// How to initialize plant control at declaration (Recommended workflow).
// [Hint]
// > All reference-variables are implemented to ease monitoring of relevant variables.
FUNCTION_BLOCK FB_Plt_Init1 EXTENDS FB_BA_View
VAR
   	{region 'Aggregates'}
		DmprSu_Open							: REFERENCE TO BOOL							REF= DmprSu.bOpen;
		DmprSu_Val							: REFERENCE TO REAL							REF= DmprSu.fActiveVal;
		DmprSu								: FB_TimerAggregateA						:= (iParent:=THIS^,					iLabel:=MyLabels.DmprSu);
		FanSu_Val							: REFERENCE TO UDINT						REF= FanSu.nActiveVal;
		FanSu								: FB_BA_AggregateM							:= (iParent:=THIS^,					iLabel:=MyLabels.FanSu);
			 
		DmprEx_Open							: REFERENCE TO BOOL							REF= DmprEx.bOpen;
		DmprEx_Val							: REFERENCE TO REAL							REF= DmprEx.fActiveVal;
		DmprEx								: FB_TimerAggregateA						:= (iParent:=THIS^,					iLabel:=MyLabels.DmprEx);
		FanEx_Val							: REFERENCE TO UDINT						REF= FanEx.nActiveVal;
		FanEx								: FB_BA_AggregateM							:= (iParent:=THIS^,					iLabel:=MyLabels.FanEx);
			 
		PreHtr_Proc							: REFERENCE TO BOOL							REF= PreHtr.Process.bActive;
		PreHtr_Val							: REFERENCE TO BOOL							REF= PreHtr.bActiveVal;
		PreHtr								: FB_ProcAggregateB							:= (iParent:=THIS^,					iLabel:=MyLabels.PreHtr,			Process:=(iLabel:=MyLabels.ProcPreRinse));
		Erc_Val								: REFERENCE TO BOOL							REF= Erc.bActiveVal;
		Erc									: FB_BA_AggregateB							:= (iParent:=THIS^,					iLabel:=MyLabels.Erc);
		Col_Val								: REFERENCE TO BOOL							REF= Col.bActiveVal;
		Col									: FB_BA_AggregateB							:= (iParent:=THIS^,					iLabel:=MyLabels.Col);
	{endregion}
	{region 'Plant'} 
		OpMode								: E_OpMod_AC								:= E_OpMod_AC.eOff;
		PlantCtrl_OpSta						: REFERENCE TO BOOL							REF= PlantCtrl.bOpSta;
		PlantCtrl_On						: REFERENCE TO BOOL							REF= PlantCtrl.bOn;
		PlantCtrl_PrVal						: REFERENCE TO UDINT						REF= PlantCtrl.nPresentValue;
		PlantCtrl_Step						: REFERENCE TO STRING						REF= PlantCtrl.sStep;
		PlantCtrl							: FB_BA_PlantCtrl := (
												iParent									:= THIS^,
												iLabel									:= MyLabels.PltCtrl,
												stOperation := (
													aOpMode								:= [ E_OpMod_AC.eDisturb,				E_OpMod_AC.eSmokeExtract,		E_OpMod_AC.eOff,			E_OpMod_AC.eOn,				E_OpMod_AC.eNightCool ],
													aPriority							:= [ E_BA_Priority.eCritical,			E_BA_Priority.eLifeSafety,		E_BA_Priority.eProgram,		E_BA_Priority.eProgram,		E_BA_Priority.eProgram ],
													aIgnoreFlags						:= [ E_BA_AggregateIgnoreFlags.Delay,	E_BA_AggregateIgnoreFlags.All,	0,							0,							0 ],
													aAggregates := [(
														iReference						:= DmprSu,
														aAggMode						:= [ 0,									100,							0,							100,						100 ]
													), (
														iReference						:= DmprEx,
														aAggMode						:= [ 0,									100,							0,							100,						100 ]
													), (
														iReference						:= PreHtr,
														aAggMode						:= [ E_OpMod_Binary.eOff,				E_OpMod_Binary.eOn,				E_OpMod_Binary.eOff,		E_OpMod_Binary.eOn,			E_OpMod_Binary.eOff ],
														bWaitForProcesses				:= TRUE
													), (
														iReference						:= Erc,
														aAggMode						:= [ E_OpMod_Binary.eOff,				E_OpMod_Binary.eOn,				E_OpMod_Binary.eOff,		E_OpMod_Binary.eOn,			E_OpMod_Binary.eOff ]
													), (
														iReference						:= Col,
														aAggMode						:= [ E_OpMod_Binary.eOff,				E_OpMod_Binary.eOn,				E_OpMod_Binary.eOff,		E_OpMod_Binary.eOn,			E_OpMod_Binary.eOff ]
													), (
														iReference						:= FanSu,
														aAggMode						:= [ E_OpMod_Step2.eOff,				E_OpMod_Step2.eStep2,			E_OpMod_Step2.eOff,			E_OpMod_Step2.eStep1,		E_OpMod_Step2.eStep2 ],
														tDelayStepDown					:= T#0S,
														tDelayStepUp					:= T#5S
													), (
														iReference						:= FanEx,
														aAggMode						:= [ E_OpMod_Step2.eOff,				E_OpMod_Step2.eStep2,			E_OpMod_Step2.eOff,			E_OpMod_Step2.eStep1,		E_OpMod_Step2.eStep2 ],
														tDelayStepDown					:= T#5S,
														tDelayStepUp					:= T#0S
													)]
											));
	{endregion}
END_VAR

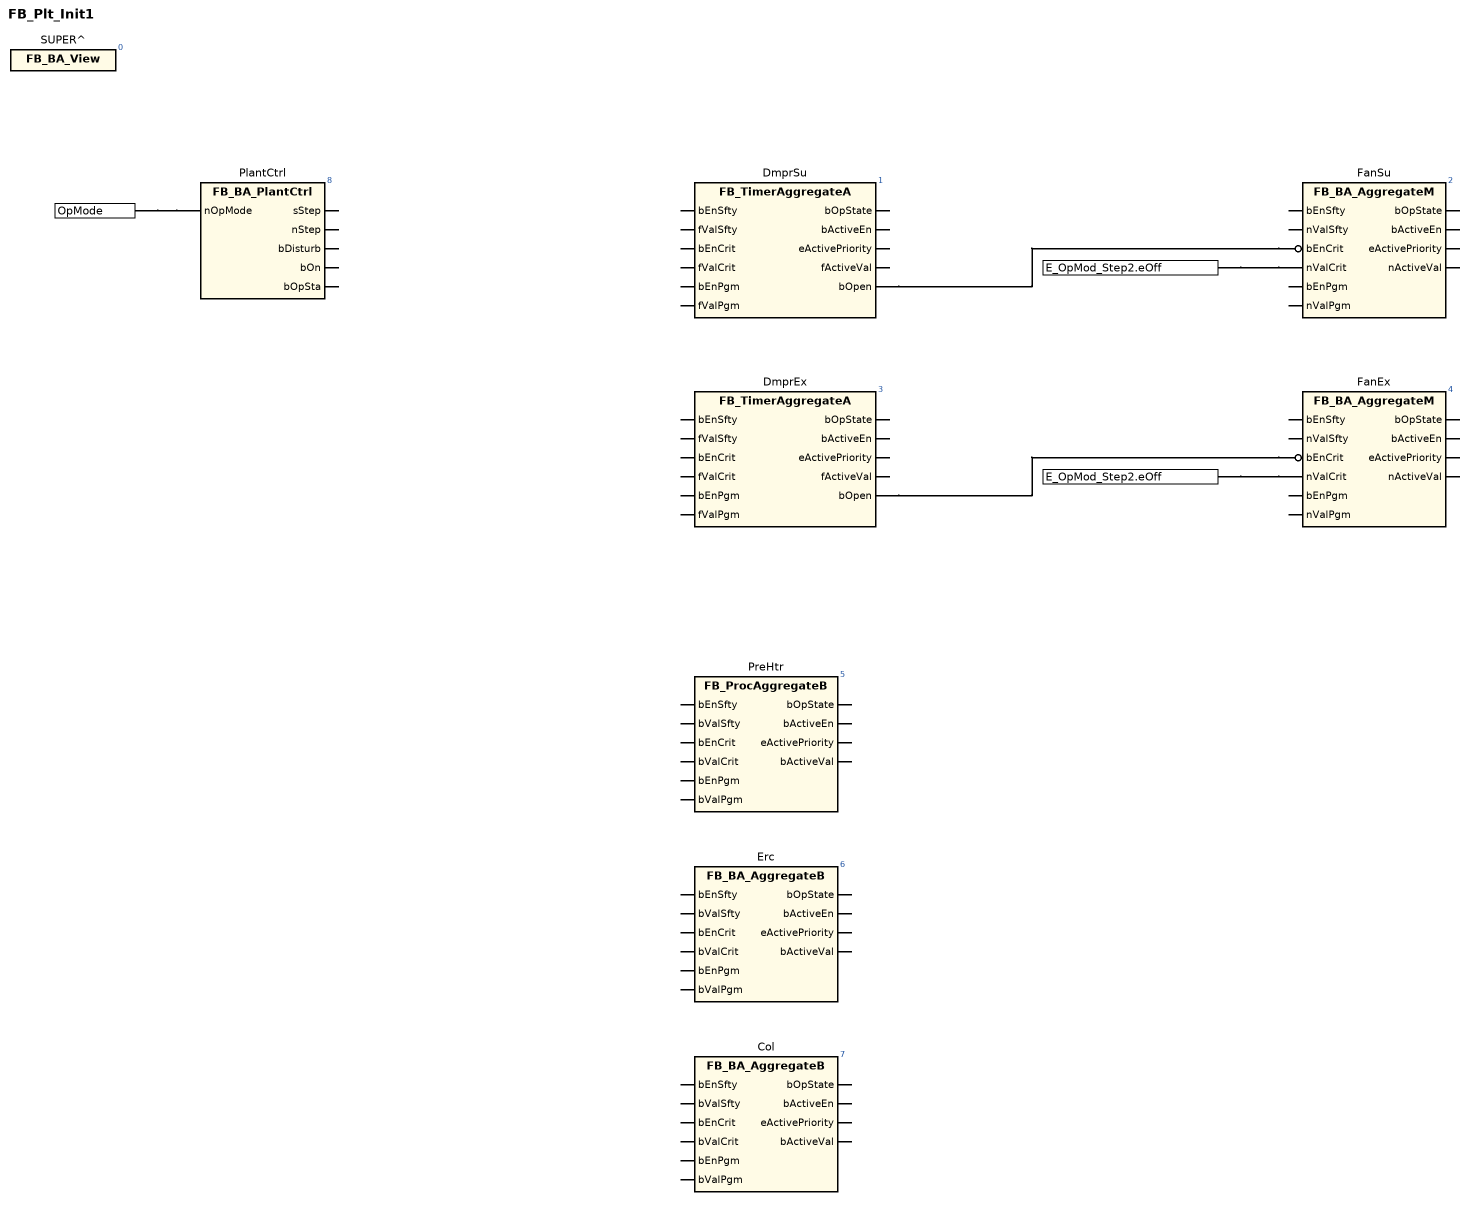
SUPER^(); // FB_BA_View
DmprSu(); // FB_TimerAggregateA
FanSu(bEnCrit := NOT DmprSu.bOpen, nValCrit := E_OpMod_Step2.eOff); // FB_BA_AggregateM
DmprEx(); // FB_TimerAggregateA
FanEx(bEnCrit := NOT DmprEx.bOpen, nValCrit := E_OpMod_Step2.eOff); // FB_BA_AggregateM
PreHtr(); // FB_ProcAggregateB
Erc(); // FB_BA_AggregateB
Col(); // FB_BA_AggregateB
PlantCtrl(nOpMode := OpMode); // FB_BA_PlantCtrl

END_FUNCTION_BLOCK

(* stored: Version 1.1.0.1, ProductVersion 3.1.4024.9
   POU FB_Plt_Init1: Id {a9ce6917-417d-453a-ad36-bec8d12e7989}, SpecialFunc None *)
